// TIA Portal project "Светофор" (V15)

(* hardware
DEVICE "S7-1200 station_1"  S7-1200 Station
   slot 0: "Rack_0"  S7-1200 Rack  Rack  V1.0
   slot 1: "PLC_1"  CPU 1215C DC/DC/DC  6ES7 215-1AG40-0XB0  V4.2
   slot 2: "AI 8x13BIT_1"  6ES7 231-4HF32-0XB0  V2.0
   slot 3: "CB 1241 (RS485)"  CB 1241 (RS485)  6ES7 241-1CH30-1XB0  V1.0
DEVICE "CSM"  SCALANCE X-Station
   slot 0: "SCALANCE X rack"  Rail
   slot 0: "Switch_1"  6GK7 277-1AA10-0AA0
*)

// ===== PLC "PLC_1"  CPU 1215C DC/DC/DC =====

VAR_GLOBAL   // PLC tag table "Default tag table"
   "System_Byte" AT %MB100 : Byte;
   "FirstScan" AT %M100.0 : Bool;
   "DiagStatusUpdate" AT %M100.1 : Bool;
   "AlwaysTRUE" AT %M100.2 : Bool;
   "AlwaysFALSE" AT %M100.3 : Bool;
   "Clock_Byte" AT %MB101 : Byte;
   "Clock_10Hz" AT %M101.0 : Bool;
   "Clock_5Hz" AT %M101.1 : Bool;
   "Clock_2.5Hz" AT %M101.2 : Bool;
   "Clock_2Hz" AT %M101.3 : Bool;
   "Clock_1.25Hz" AT %M101.4 : Bool;
   "Clock_1Hz" AT %M101.5 : Bool;
   "Clock_0.625Hz" AT %M101.6 : Bool;
   "Clock_0.5Hz" AT %M101.7 : Bool;
   "Транспортный датчик 1" AT %M0.0 : Bool;
   "Транспортный датчик 2" AT %M0.1 : Bool;
   "Зеленый Транспорт HL3" AT %Q0.0 : Bool;
   "Желтый Транспорт HL2" AT %Q0.1 : Bool;
   "Красный Транспорт HL1" AT %Q0.2 : Bool;
   "Красный Пешеход HL4" AT %Q0.3 : Bool;
   "Зеленый Пешеход HL5" AT %Q0.4 : Bool;
   "Звуковой Сигнализатор BA1 BA2" AT %Q0.5 : Bool;
   "Датчик пешеходов SQ1" AT %I0.0 : Bool;
   "Датчик пешеходов SQ2" AT %I0.1 : Bool;
   "Сенсорное табло SQ3" AT %I0.2 : Bool;
   "Сенсорное табло SQ4" AT %I0.3 : Bool;
   "Сенсорное табло SQ5" AT %I0.4 : Bool;
   "ШАГ" AT %MW1 : Int;
   "Режим зеленой волны" AT %M0.3 : Bool;
   "n" AT %MW3 : Int;
   "Ошибка" AT %M0.4 : Bool;
   "Сброс ошибки" AT %M0.5 : Bool;
   "Проверка +1" AT %M0.6 : Bool;
   "Записывать ошибки в отчет" AT %M0.7 : Bool;
END_VAR

DATA_BLOCK "Data_block_1"   // DB3
{ S7_Optimized_Access := 'TRUE' }
VERSION : 0.1
   VAR
      "Load done" : Bool;
      "Load Error" : Bool;
      "Load Status" : Word;
      "Master done" : Bool;
      "Master Busy" : Bool;
      "Master Error" : Bool;
      "Master Status" : Word;
   END_VAR
BEGIN
END_DATA_BLOCK

DATA_BLOCK "ArcenCrossData"   // DB4
{ S7_Optimized_Access := 'FALSE' }
VERSION : 0.1
   VAR
      data : Array[0..16] of Int;
   END_VAR
BEGIN
   // data[0] : Контр.Сумма тела
   // data[1] : Данные
   // data[2] : Данные
   // data[3] : Неизменное
END_DATA_BLOCK

DATA_BLOCK "Data_block_2"   // DB6
{ S7_Optimized_Access := 'TRUE' }
VERSION : 0.1
   VAR
      "Load done" : Bool;
      "Load Error" : Bool;
      "Load Status" : Word;
      "Master done" : Bool;
      "Master Busy" : Bool;
      "Master Error" : Bool;
      "Master Status" : Word;
   END_VAR
BEGIN
END_DATA_BLOCK

DATA_BLOCK "ArcenCrossData2"   // DB8
{ S7_Optimized_Access := 'FALSE' }
VERSION : 0.1
   VAR
      data : Array[0..16] of Int;
   END_VAR
BEGIN
   // data[0] : Контр.Сумма тела
   // data[1] : Данные
   // data[2] : Данные
   // data[3] : Неизменное
END_DATA_BLOCK

DATA_BLOCK "Data_block_3"   // DB17
{ S7_Optimized_Access := 'TRUE' }
VERSION : 0.1
   VAR
      Records : UDInt := 25;
      "name" : String := 'logging';
      id : DWord := 1;
      header : String := 'Error';
      done : Bool;
      data : Struct
         "current error" : String := 'Number of checks exceeded';
      END_STRUCT;
   END_VAR
BEGIN
END_DATA_BLOCK

// folder: System blocks/Program resources

DATA_BLOCK "IEC_Timer_0_DB"   // DB9
{ S7_Optimized_Access := 'TRUE' }
AUTHOR : Simatic
FAMILY : IEC
NAME : IEC_TMR
VERSION : 1.0
// stored: InstanceOfName IEC_TIMER
"IEC_TIMER"
BEGIN
END_DATA_BLOCK

DATA_BLOCK "IEC_Timer_0_DB_1"   // DB10
{ S7_Optimized_Access := 'TRUE' }
AUTHOR : Simatic
FAMILY : IEC
NAME : IEC_TMR
VERSION : 1.0
// stored: InstanceOfName IEC_TIMER
"IEC_TIMER"
BEGIN
END_DATA_BLOCK

DATA_BLOCK "IEC_Timer_0_DB_2"   // DB11
{ S7_Optimized_Access := 'TRUE' }
AUTHOR : Simatic
FAMILY : IEC
NAME : IEC_TMR
VERSION : 1.0
// stored: InstanceOfName IEC_TIMER
"IEC_TIMER"
BEGIN
END_DATA_BLOCK

DATA_BLOCK "IEC_Timer_0_DB_3"   // DB12
{ S7_Optimized_Access := 'TRUE' }
AUTHOR : Simatic
FAMILY : IEC
NAME : IEC_TMR
VERSION : 1.0
// stored: InstanceOfName IEC_TIMER
"IEC_TIMER"
BEGIN
END_DATA_BLOCK

DATA_BLOCK "IEC_Timer_0_DB_4"   // DB13
{ S7_Optimized_Access := 'TRUE' }
AUTHOR : Simatic
FAMILY : IEC
NAME : IEC_TMR
VERSION : 1.0
// stored: InstanceOfName IEC_TIMER
"IEC_TIMER"
BEGIN
END_DATA_BLOCK

DATA_BLOCK "IEC_Timer_0_DB_5"   // DB14
{ S7_Optimized_Access := 'TRUE' }
AUTHOR : Simatic
FAMILY : IEC
NAME : IEC_TMR
VERSION : 1.0
// stored: InstanceOfName IEC_TIMER
"IEC_TIMER"
BEGIN
END_DATA_BLOCK

DATA_BLOCK "IEC_Counter_0_DB"   // DB15
{ S7_Optimized_Access := 'TRUE' }
AUTHOR : Simatic
FAMILY : IEC
NAME : CNTR
VERSION : 1.0
// stored: InstanceOfName IEC_COUNTER
"IEC_COUNTER"
BEGIN
END_DATA_BLOCK

// folder: (top level)

ORGANIZATION_BLOCK "Main"   // OB1, LAD, ProgramCycle
TITLE = "Main Program Sweep (Cycle)"
{ S7_Optimized_Access := 'TRUE' }
VERSION : 0.1
   VAR_INPUT
      Initial_Call : Bool;   // Initial call of this OB
      Remanence : Bool;   // =True, if remanent data are available
   END_VAR
   VAR_TEMP
      D1 : Bool;
   END_VAR
   VAR_TEMP   // added for the SCL form of the ladder/FBD networks
      _w1 : Bool;
      _w2 : Bool;
   END_VAR
BEGIN

REGION Network 1: Проверка Транспортных светофоров
   // Проверка Транспортных светофоров
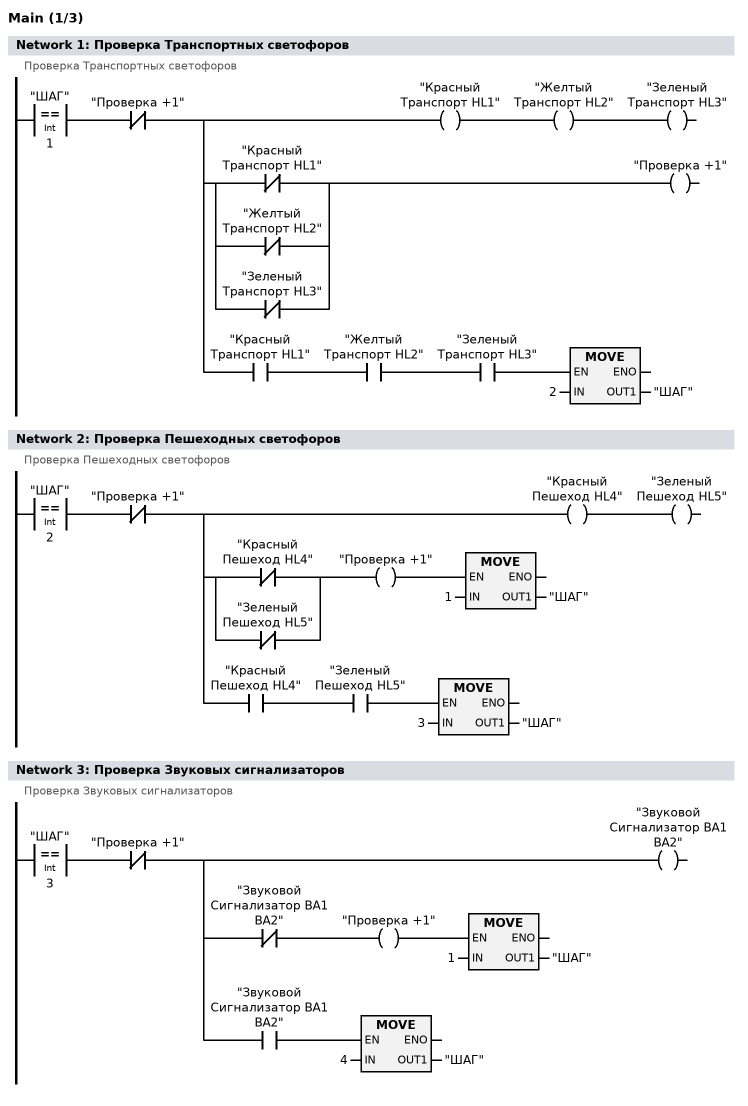
   RUNG wire#powerrail
      { S7_Templates := "SrcType := Int" } EQ_Contact(in1 := "ШАГ", in2 := 1)
      I_Contact( "Проверка +1" )
      wire#w1
      Coil( "Красный Транспорт HL1" )
      Coil( "Желтый Транспорт HL2" )
      Coil( "Зеленый Транспорт HL3" )
   END_RUNG
   RUNG wire#w1
      I_Contact( "Красный Транспорт HL1" )
      wire#w2
      Coil( "Проверка +1" )
   END_RUNG
   RUNG wire#w1
      I_Contact( "Желтый Транспорт HL2" )
   END_RUNG wire#w2
   RUNG wire#w1
      I_Contact( "Зеленый Транспорт HL3" )
   END_RUNG wire#w2
   RUNG wire#w1
      Contact( "Красный Транспорт HL1" )
      Contact( "Желтый Транспорт HL2" )
      Contact( "Зеленый Транспорт HL3" )
      Move(in := 2, out1 => "ШАГ")
   END_RUNG
   // the same network as SCL:
   "Красный Транспорт HL1" := ("ШАГ" = 1) AND NOT "Проверка +1";
   "Желтый Транспорт HL2" := "Красный Транспорт HL1";
   "Зеленый Транспорт HL3" := "Красный Транспорт HL1";
   "Проверка +1" := "Красный Транспорт HL1" AND (NOT "Красный Транспорт HL1" OR NOT "Желтый Транспорт HL2" OR NOT "Зеленый Транспорт HL3");
   IF "Красный Транспорт HL1" AND "Красный Транспорт HL1" AND "Желтый Транспорт HL2" AND "Зеленый Транспорт HL3" THEN
       "ШАГ" := 2;
   END_IF;
END_REGION

REGION Network 2: Проверка Пешеходных светофоров
   // Проверка Пешеходных светофоров
   RUNG wire#powerrail
      { S7_Templates := "SrcType := Int" } EQ_Contact(in1 := "ШАГ", in2 := 2)
      I_Contact( "Проверка +1" )
      wire#w1
      Coil( "Красный Пешеход HL4" )
      Coil( "Зеленый Пешеход HL5" )
   END_RUNG
   RUNG wire#w1
      I_Contact( "Красный Пешеход HL4" )
      wire#w2
      Coil( "Проверка +1" )
      Move(in := 1, out1 => "ШАГ")
   END_RUNG
   RUNG wire#w1
      I_Contact( "Зеленый Пешеход HL5" )
   END_RUNG wire#w2
   RUNG wire#w1
      Contact( "Красный Пешеход HL4" )
      Contact( "Зеленый Пешеход HL5" )
      Move(in := 3, out1 => "ШАГ")
   END_RUNG
   // the same network as SCL:
   "Красный Пешеход HL4" := ("ШАГ" = 2) AND NOT "Проверка +1";
   "Зеленый Пешеход HL5" := "Красный Пешеход HL4";
   "Проверка +1" := "Красный Пешеход HL4" AND (NOT "Красный Пешеход HL4" OR NOT "Зеленый Пешеход HL5");
   IF "Проверка +1" THEN "ШАГ" := 1; END_IF;
   IF "Красный Пешеход HL4" AND "Красный Пешеход HL4" AND "Зеленый Пешеход HL5" THEN "ШАГ" := 3; END_IF;
END_REGION

REGION Network 3: Проверка Звуковых сигнализаторов
   // Проверка Звуковых сигнализаторов
   RUNG wire#powerrail
      { S7_Templates := "SrcType := Int" } EQ_Contact(in1 := "ШАГ", in2 := 3)
      I_Contact( "Проверка +1" )
      wire#w1
      Coil( "Звуковой Сигнализатор BA1 BA2" )
   END_RUNG
   RUNG wire#w1
      I_Contact( "Звуковой Сигнализатор BA1 BA2" )
      Coil( "Проверка +1" )
      Move(in := 1, out1 => "ШАГ")
   END_RUNG
   RUNG wire#w1
      Contact( "Звуковой Сигнализатор BA1 BA2" )
      Move(in := 4, out1 => "ШАГ")
   END_RUNG
   // the same network as SCL:
   "Звуковой Сигнализатор BA1 BA2" := ("ШАГ" = 3) AND NOT "Проверка +1";
   "Проверка +1" := "Звуковой Сигнализатор BA1 BA2" AND NOT "Звуковой Сигнализатор BA1 BA2";
   IF "Проверка +1" THEN "ШАГ" := 1; END_IF;
   IF "Звуковой Сигнализатор BA1 BA2" AND "Звуковой Сигнализатор BA1 BA2" THEN "ШАГ" := 4; END_IF;
END_REGION

REGION Network 4: Подсчет количества проверок
   // Подсчет количества проверок.
   // Сброс ошибки и обнуление счетчика проверок.
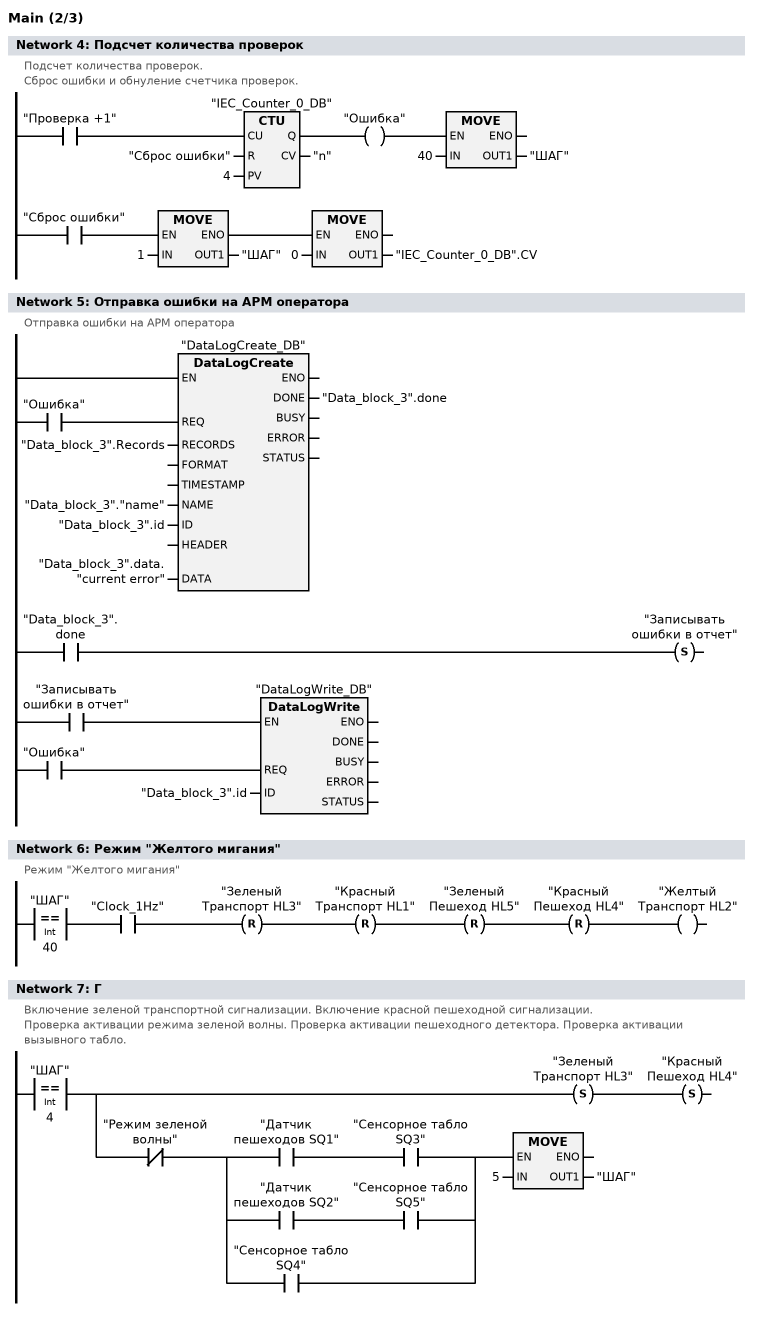
   "IEC_Counter_0_DB".CTU(CU := "Проверка +1", R := "Сброс ошибки", PV := 4, CV => "n");
   "Ошибка" := "IEC_Counter_0_DB".Q;
   IF "IEC_Counter_0_DB".Q THEN "ШАГ" := 40; END_IF;
   IF "Сброс ошибки" THEN
       "ШАГ" := 1;
       "IEC_Counter_0_DB".CV := 0;
   END_IF;
END_REGION

REGION Network 5: Отправка ошибки на АРМ оператора
   // Отправка ошибки на АРМ оператора
   "DataLogCreate_DB"(REQ := "Ошибка",   // DataLogCreate
                      RECORDS := "Data_block_3".Records,
                      "NAME" := "Data_block_3"."name",
                      ID := "Data_block_3".id,
                      DATA := "Data_block_3".data."current error",
                      DONE => "Data_block_3".done);
   IF "Data_block_3".done THEN "Записывать ошибки в отчет" := TRUE; END_IF;
   IF "Записывать ошибки в отчет" THEN
       "DataLogWrite_DB"(REQ := "Ошибка", ID := "Data_block_3".id);   // DataLogWrite
   END_IF;
END_REGION

REGION Network 6: Режим "Желтого мигания"
   // Режим "Желтого мигания"
   RUNG wire#powerrail
      { S7_Templates := "SrcType := Int" } EQ_Contact(in1 := "ШАГ", in2 := 40)
      Contact( "Clock_1Hz" )
      R_Coil( "Зеленый Транспорт HL3" )
      R_Coil( "Красный Транспорт HL1" )
      R_Coil( "Зеленый Пешеход HL5" )
      R_Coil( "Красный Пешеход HL4" )
      Coil( "Желтый Транспорт HL2" )
   END_RUNG
   // the same network as SCL:
   #_w1 := ("ШАГ" = 40) AND "Clock_1Hz";
   IF #_w1 THEN
       "Зеленый Транспорт HL3" := FALSE;
       "Красный Транспорт HL1" := FALSE;
       "Зеленый Пешеход HL5" := FALSE;
       "Красный Пешеход HL4" := FALSE;
   END_IF;
   "Желтый Транспорт HL2" := #_w1;
END_REGION

REGION Network 7: Г
   // Включение зеленой транспортной сигнализации. Включение красной пешеходной сигнализации.
   // Проверка активации режима зеленой волны. Проверка активации пешеходного детектора. Проверка активации вызывного табло.
   RUNG wire#powerrail
      { S7_Templates := "SrcType := Int" } EQ_Contact(in1 := "ШАГ", in2 := 4)
      wire#w1
      S_Coil( "Зеленый Транспорт HL3" )
      S_Coil( "Красный Пешеход HL4" )
   END_RUNG
   RUNG wire#w1
      I_Contact( "Режим зеленой волны" )
      wire#w2
      Contact( "Датчик пешеходов SQ1" )
      Contact( "Сенсорное табло SQ3" )
      wire#w3
      Move(in := 5, out1 => "ШАГ")
   END_RUNG
   RUNG wire#w2
      Contact( "Датчик пешеходов SQ2" )
      Contact( "Сенсорное табло SQ5" )
   END_RUNG wire#w3
   RUNG wire#w2
      Contact( "Сенсорное табло SQ4" )
   END_RUNG wire#w3
   // the same network as SCL:
   #_w1 := "ШАГ" = 4;
   IF #_w1 THEN
       "Зеленый Транспорт HL3" := TRUE;
       "Красный Пешеход HL4" := TRUE;
   END_IF;
   IF #_w1 AND NOT "Режим зеленой волны" AND (("Датчик пешеходов SQ1" AND "Сенсорное табло SQ3") OR ("Датчик пешеходов SQ2" AND "Сенсорное табло SQ5") OR "Сенсорное табло SQ4") THEN
       "ШАГ" := 5;
   END_IF;
END_REGION

REGION Network 8: Д
   // Переменное включение/выключение транспортной зеленой сигнализации в течении пяти секунд с интервалом в одну секунду.
   // Включение транспортной желтой сигнализации в течении трех секунд. Включение транспортной красной сигнализации.
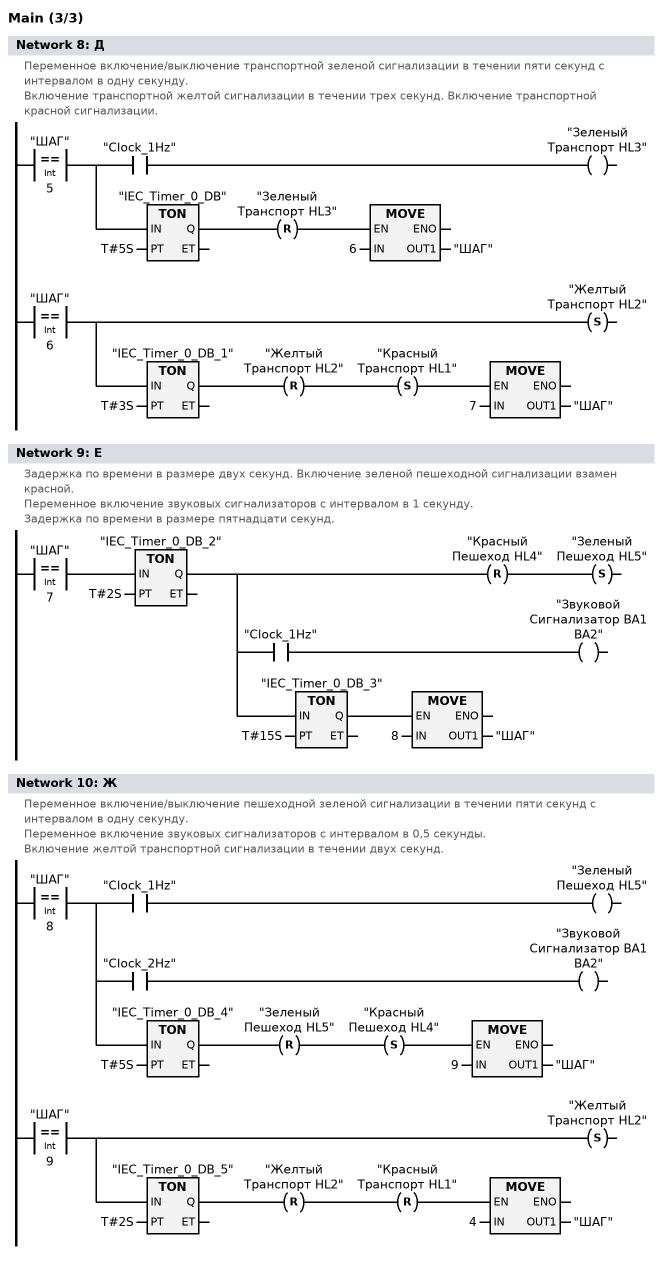
   #_w1 := "ШАГ" = 5;
   "Зеленый Транспорт HL3" := #_w1 AND "Clock_1Hz";
   "IEC_Timer_0_DB".TON(IN := #_w1, PT := T#5S);
   IF "IEC_Timer_0_DB".Q THEN
       "Зеленый Транспорт HL3" := FALSE;
       "ШАГ" := 6;
   END_IF;
   #_w2 := "ШАГ" = 6;
   IF #_w2 THEN "Желтый Транспорт HL2" := TRUE; END_IF;
   "IEC_Timer_0_DB_1".TON(IN := #_w2, PT := T#3S);
   IF "IEC_Timer_0_DB_1".Q THEN
       "Желтый Транспорт HL2" := FALSE;
       "Красный Транспорт HL1" := TRUE;
       "ШАГ" := 7;
   END_IF;
END_REGION

REGION Network 9: Е
   // Задержка по времени в размере двух секунд. Включение зеленой пешеходной сигнализации взамен красной.
   // Переменное включение звуковых сигнализаторов с интервалом в 1 секунду.
   // Задержка по времени в размере пятнадцати секунд.
   "IEC_Timer_0_DB_2".TON(IN := "ШАГ" = 7, PT := T#2S);
   IF "IEC_Timer_0_DB_2".Q THEN
       "Красный Пешеход HL4" := FALSE;
       "Зеленый Пешеход HL5" := TRUE;
   END_IF;
   "Звуковой Сигнализатор BA1 BA2" := "IEC_Timer_0_DB_2".Q AND "Clock_1Hz";
   "IEC_Timer_0_DB_3".TON(IN := "IEC_Timer_0_DB_2".Q, PT := T#15S);
   IF "IEC_Timer_0_DB_3".Q THEN "ШАГ" := 8; END_IF;
END_REGION

REGION Network 10: Ж
   // Переменное включение/выключение пешеходной зеленой сигнализации в течении пяти секунд с интервалом в одну секунду.
   // Переменное включение звуковых сигнализаторов с интервалом в 0,5 секунды.
   // Включение желтой транспортной сигнализации в течении двух секунд.
   #_w1 := "ШАГ" = 8;
   "Зеленый Пешеход HL5" := #_w1 AND "Clock_1Hz";
   "Звуковой Сигнализатор BA1 BA2" := #_w1 AND "Clock_2Hz";
   "IEC_Timer_0_DB_4".TON(IN := #_w1, PT := T#5S);
   IF "IEC_Timer_0_DB_4".Q THEN
       "Зеленый Пешеход HL5" := FALSE;
       "Красный Пешеход HL4" := TRUE;
       "ШАГ" := 9;
   END_IF;
   #_w2 := "ШАГ" = 9;
   IF #_w2 THEN "Желтый Транспорт HL2" := TRUE; END_IF;
   "IEC_Timer_0_DB_5".TON(IN := #_w2, PT := T#2S);
   IF "IEC_Timer_0_DB_5".Q THEN
       "Желтый Транспорт HL2" := FALSE;
       "Красный Транспорт HL1" := FALSE;
       "ШАГ" := 4;
   END_IF;
END_REGION
END_ORGANIZATION_BLOCK

ORGANIZATION_BLOCK "Cyclic interrupt"   // OB30, LAD, CyclicInterrupt
{ S7_Optimized_Access := 'TRUE' }
VERSION : 0.1
   VAR_INPUT
      Initial_Call : Bool;   // Initial call of this OB
      Event_Count : Int;   // Events discarded
   END_VAR
BEGIN

REGION Network 1: Аркен кросс №1
   // подключение к датчику Аркен кросс №1
   // Чтение данных с датчика
   // Обнаружение транспорта
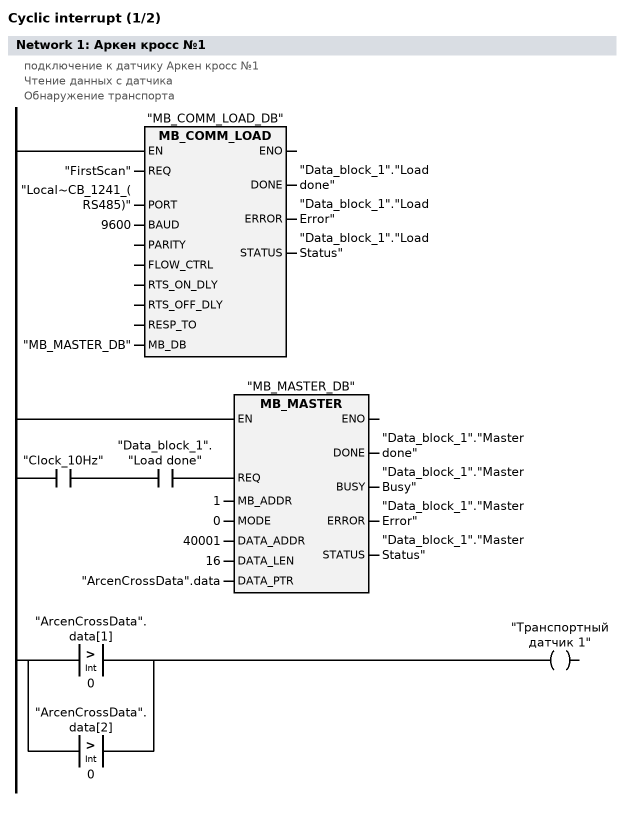
   "MB_COMM_LOAD_DB"(REQ := "FirstScan",   // MB_COMM_LOAD
                     PORT := "Local~CB_1241_(RS485)",
                     BAUD := 9600,
                     MB_DB := "MB_MASTER_DB",
                     DONE => "Data_block_1"."Load done",
                     ERROR => "Data_block_1"."Load Error",
                     STATUS => "Data_block_1"."Load Status");
   "MB_MASTER_DB"(REQ := "Clock_10Hz" AND "Data_block_1"."Load done",   // MB_MASTER
                  MB_ADDR := 1,
                  MODE := 0,
                  DATA_ADDR := 40001,
                  DATA_LEN := 16,
                  DATA_PTR := "ArcenCrossData".data,
                  DONE => "Data_block_1"."Master done",
                  BUSY => "Data_block_1"."Master Busy",
                  ERROR => "Data_block_1"."Master Error",
                  STATUS => "Data_block_1"."Master Status");
   "Транспортный датчик 1" := ("ArcenCrossData".data[1] > 0) OR ("ArcenCrossData".data[2] > 0);
END_REGION

REGION Network 2: Аркен кросс №2
   // подключение к датчику Аркен кросс №2
   // Чтение данных с датчика
   // Обнаружение транспорта
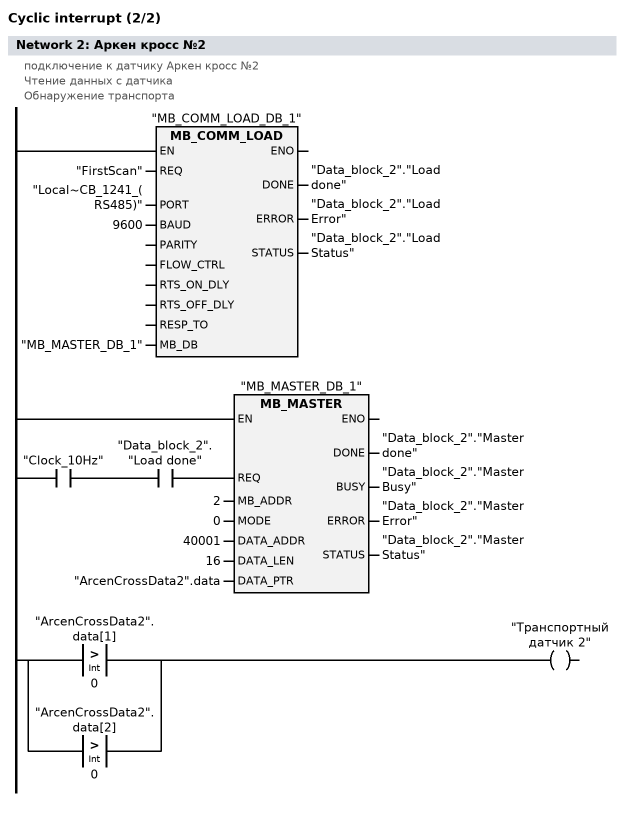
   "MB_COMM_LOAD_DB_1"(REQ := "FirstScan",   // MB_COMM_LOAD
                       PORT := "Local~CB_1241_(RS485)",
                       BAUD := 9600,
                       MB_DB := "MB_MASTER_DB_1",
                       DONE => "Data_block_2"."Load done",
                       ERROR => "Data_block_2"."Load Error",
                       STATUS => "Data_block_2"."Load Status");
   "MB_MASTER_DB_1"(REQ := "Clock_10Hz" AND "Data_block_2"."Load done",   // MB_MASTER
                    MB_ADDR := 2,
                    MODE := 0,
                    DATA_ADDR := 40001,
                    DATA_LEN := 16,
                    DATA_PTR := "ArcenCrossData2".data,
                    DONE => "Data_block_2"."Master done",
                    BUSY => "Data_block_2"."Master Busy",
                    ERROR => "Data_block_2"."Master Error",
                    STATUS => "Data_block_2"."Master Status");
   "Транспортный датчик 2" := ("ArcenCrossData2".data[1] > 0) OR ("ArcenCrossData2".data[2] > 0);
END_REGION
END_ORGANIZATION_BLOCK

ORGANIZATION_BLOCK "Startup"   // OB100, LAD, Startup
TITLE = "Complete Restart"
{ S7_Optimized_Access := 'TRUE' }
VERSION : 0.1
   VAR_INPUT
      LostRetentive : Bool;   // True if retentive data are lost
      LostRTC : Bool;   // True if date and time are lost
   END_VAR
BEGIN

REGION Network 1: Установка значений по умолчанию при запуске контроллера
   // Шаг = 1. Количество проверок = 0.
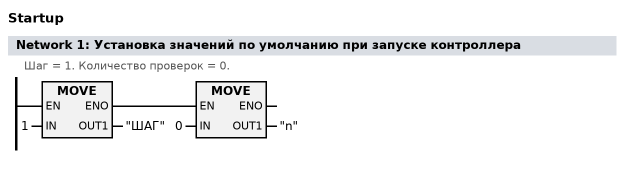
   RUNG wire#powerrail
      Move(in := 1, out1 => "ШАГ")
      Move(in := 0, out1 => "n")
   END_RUNG
   // the same network as SCL:
   "ШАГ" := 1;
   "n" := 0;
END_REGION
END_ORGANIZATION_BLOCK